{region '#Template'}
	{attribute 'Version' := '1.2.1.0'}
	{attribute 'Tags' := '"LCID": "1031", "Text": "Universal, Control, Timer"'}
	{attribute 'Tags' := '"LCID": "1033", "Text": "Universal, Control, Timer"'}
	{attribute 'Using' := '"Type": "Template", "URI": "BA2_Param"'}
	{attribute 'Description' := '"LCID": "1031", "Text": "Zeitglied Einschaltverzögert"'}
	{attribute 'Description' := '"LCID": "1033", "Text": "Timer switch-on delayed"'}
{endregion}
FUNCTION_BLOCK FB_BA_DlyOn EXTENDS FB_BA_View
VAR_INPUT
	bVal					: BOOL;	
END_VAR
VAR_OUTPUT
	bQ						: BOOL;
	nRT						: UDINT;// Restzeit [s] // remaining time [s]	
END_VAR
VAR_INPUT CONSTANT
	TiDly					: FB_BA_AV_Op;		
END_VAR	
VAR	
	tonDlyOn				: TON;
END_VAR
VAR // added by the converter: edge detectors and wires of the graphical bodies
    _w1, _w2 : ANY;
END_VAR

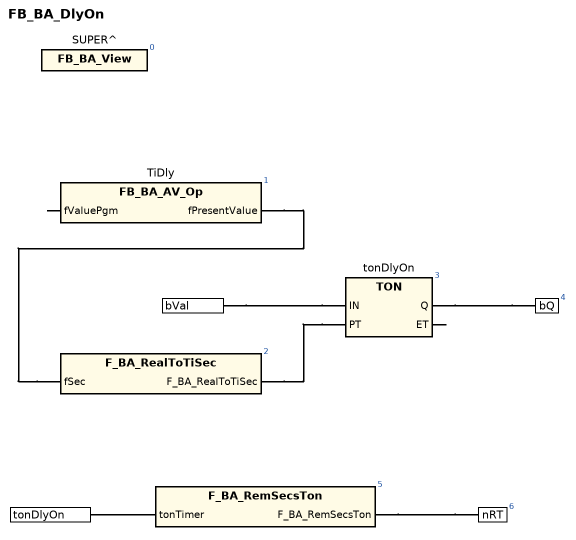
SUPER^(); // FB_BA_View
TiDly(); // FB_BA_AV_Op
_w1 := F_BA_RealToTiSec(fSec := TiDly.fPresentValue);
tonDlyOn(IN := bVal, PT := _w1); // TON
bQ := tonDlyOn.Q;
_w2 := F_BA_RemSecsTon(tonTimer := tonDlyOn);
nRT := _w2;

METHOD FB_init : BOOL
VAR_INPUT
	bInitRetains : BOOL; // if TRUE, the retain variables are initialized (warm start / cold start)
	bInCopyCode : BOOL;  // if TRUE, the instance afterwards gets moved into the copy code (online change)
END_VAR
TiDly.iParent			:= THIS^;
TiDly.iLabel			:= LblUniControl.DelayOn_TiDly;		 
TiDly.sObjectName		:= '{Idx=01}';								 	 
TiDly.eUnit 			:= E_BA_Unit.eTime_Seconds;								 
TiDly.fValueRm			:= 0;		
TiDly.fCOVIncrement		:= BA2_Param.fDefCOVIncrement;
END_METHOD

END_FUNCTION_BLOCK

(* stored: Version 1.1.0.1, ProductVersion 3.1.4024.9
   POU FB_BA_DlyOn: Id {5abcdfe0-b03d-47fc-9dc0-db83fa2785df}, SpecialFunc None
   Method FB_init: Id {00cc2adc-40dd-4c51-9fd1-7e8123212515} *)
